INTERFACE I_DictionaryItem EXTENDS I_LinkedListItem_ReadWrite

END_INTERFACE

(* stored: Version 1.1.0.1, ProductVersion 3.1.4024.12
   Itf I_DictionaryItem: Id {8fcac613-23cc-4863-9d10-212414021dda} *)
